// Implicitly generated code : DO NOT EDIT
FUNCTION CheckRangeUnsigned : UDINT
VAR_INPUT
	value, lower, upper: UDINT;
END_VAR

// Implicitly generated code : Only an Implementation suggestion
IF (value < lower) THEN
	CheckRangeUnsigned := lower;
	gvlChecks.dCheckRangeUnsigned := gvlChecks.dCheckRangeUnsigned + 1;
ELSIF(value > upper) THEN
	CheckRangeUnsigned := upper;
	gvlChecks.dCheckRangeUnsigned := gvlChecks.dCheckRangeUnsigned + 1;
ELSE
	CheckRangeUnsigned := value;
END_IF

END_FUNCTION

(* stored: Version 1.1.0.1, ProductVersion 3.1.4026.13, FileIdentifier 268568911dcdd7393794681e037ba3686917a179, FileSignature a2f1f8b77c2d2b02d769b31b0a9daed70e10cea2af5580c4ff1aa64a377f63daa26976c9278552f0e2e6880ee43394731929767ae5f07eb383e89d9eac750e7c8aa9f8d116063dae35c973f508562a0121aab721fde0675e2311718769380cd69437341b28fe6253ca9f785b1f013c814599e6ead4af22893ba886be5f48248cc865b3f3275c96f9eaf42124c4d068effa3fbef4ac92006f13dc837b6292f53ce6bb834a476227a9fa157eb78741739a327c04f8a48bb175b6aa055f4187fc3d22ea35dad1e2f355fb48de038a6eca3a13d90b923ff88d62654f387e2fe9242b8aed9c6306baa8f41cea2f98315295a8a52d217e424352326632795130cfddd7
   POU CheckRangeUnsigned: Id {36bf99f8-15d6-410e-b338-663fb75109d2}, SpecialFunc CheckRangeUnsigned *)
